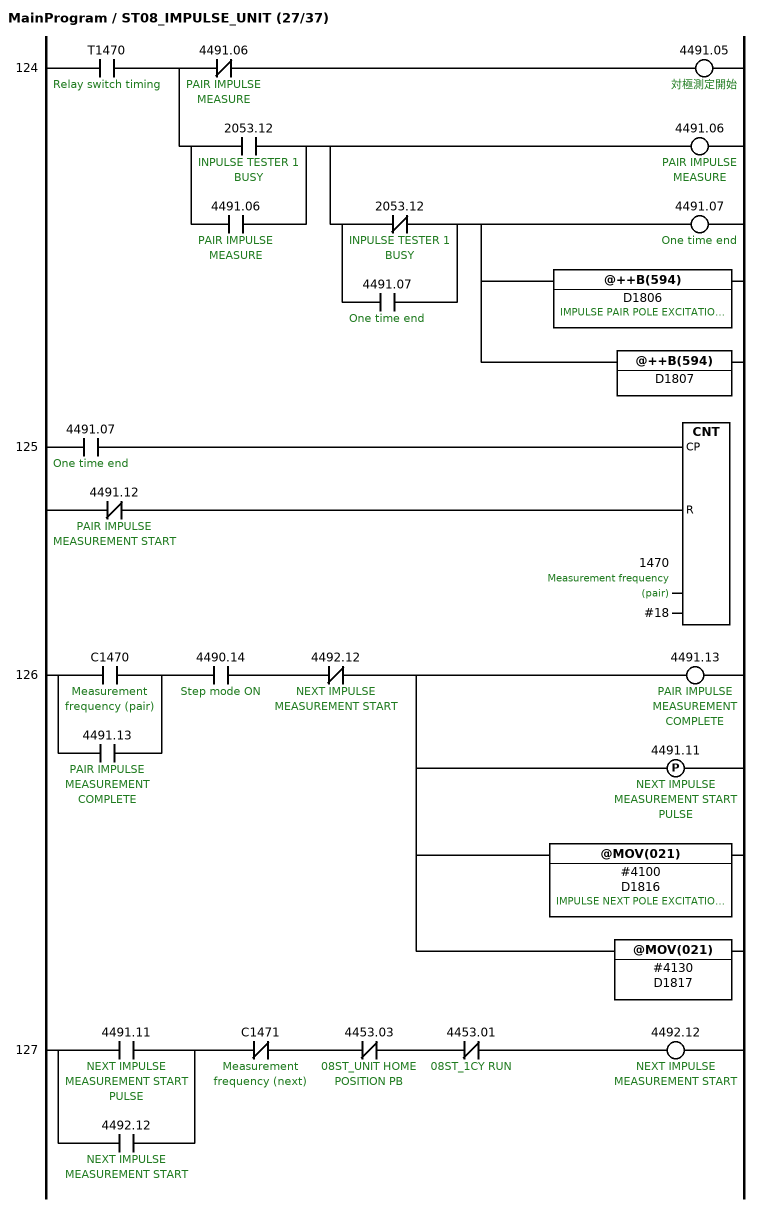
; [picture p456: MainProgram / ST08_IMPULSE_UNIT, rungs 124-127]
; rung 124
LD T1470  ; Relay switch timing
OUT TR0
ANDNOT 4491.06  ; PAIR IMPULSE MEASURE
OUT 4491.05  ; 対極測定開始
LD TR0
LD 2053.12  ; INPULSE TESTER 1 BUSY
OR 4491.06  ; PAIR IMPULSE MEASURE
ANDLD
OUT 4491.06  ; PAIR IMPULSE MEASURE
LDNOT 2053.12  ; INPULSE TESTER 1 BUSY
OR 4491.07  ; One time end
ANDLD
OUT 4491.07  ; One time end
@++B(594) D1806  ; IMPULSE PAIR POLE EXCITATION PATTERN DM STORING(INDIVIDUAL)
@++B(594) D1807
; rung 125
LD 4491.07  ; One time end
LDNOT 4491.12  ; PAIR IMPULSE MEASUREMENT START
CNT 1470 #18  ; Measurement frequency (pair)  // 6 => 18
; rung 126
LD C1470  ; Measurement frequency (pair)
OR 4491.13  ; PAIR IMPULSE MEASUREMENT COMPLETE
AND 4490.14  ; Step mode ON
ANDNOT 4492.12  ; NEXT IMPULSE MEASUREMENT START
OUT 4491.13  ; PAIR IMPULSE MEASUREMENT COMPLETE
DIFU(013) 4491.11  ; NEXT IMPULSE MEASUREMENT START PULSE
@MOV(021) #4100 D1816  ; IMPULSE NEXT POLE EXCITATION PATTERN DM STORING(INDIVIDUAL)
@MOV(021) #4130 D1817
; rung 127
LD 4491.11  ; NEXT IMPULSE MEASUREMENT START PULSE
OR 4492.12  ; NEXT IMPULSE MEASUREMENT START
ANDNOT C1471  ; Measurement frequency (next)
ANDNOT 4453.03  ; 08ST_UNIT HOME POSITION PB
ANDNOT 4453.01  ; 08ST_1CY RUN
OUT 4492.12  ; NEXT IMPULSE MEASUREMENT START

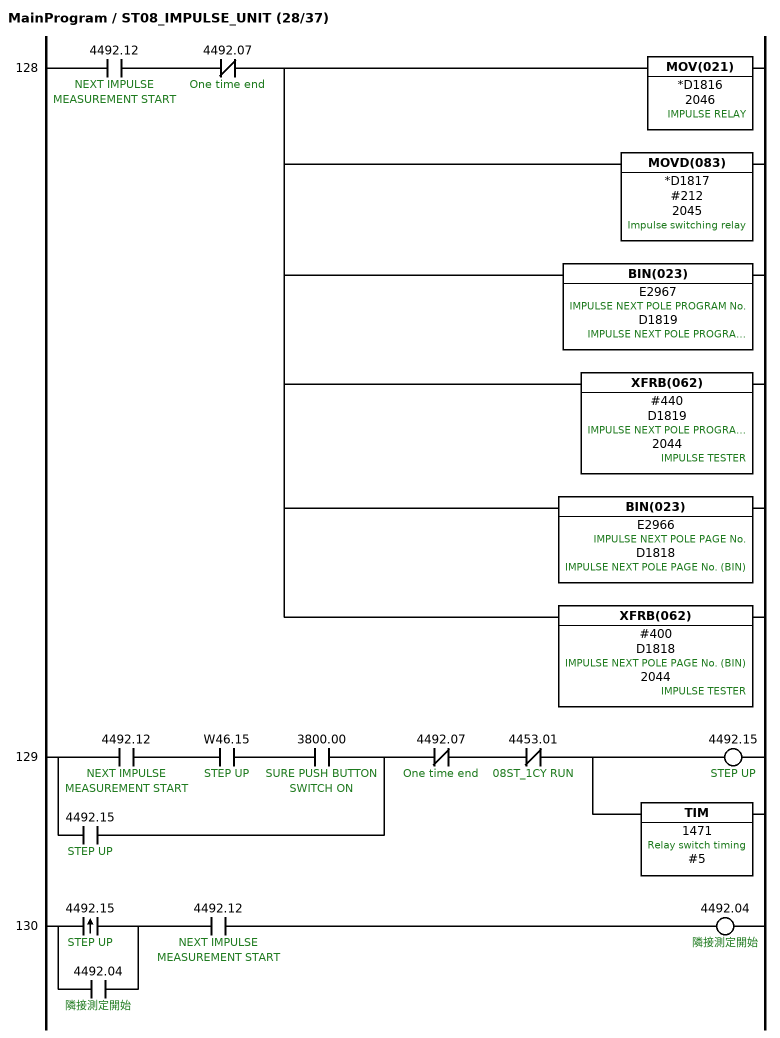
; rung 128
LD 4492.12  ; NEXT IMPULSE MEASUREMENT START
ANDNOT 4492.07  ; One time end
MOV(021) *D1816 2046  ; IMPULSE RELAY
MOVD(083) *D1817 #212 2045  ; Impulse switching relay
BIN(023) E2967 D1819  ; IMPULSE NEXT POLE PROGRAM No., IMPULSE NEXT POLE PROGRAM No.(BIN)
XFRB(062) #440 D1819 2044  ; IMPULSE NEXT POLE PROGRAM No.(BIN), IMPULSE TESTER
BIN(023) E2966 D1818  ; IMPULSE NEXT POLE PAGE No., IMPULSE NEXT POLE PAGE No. (BIN)
XFRB(062) #400 D1818 2044  ; IMPULSE NEXT POLE PAGE No. (BIN), IMPULSE TESTER
; rung 129
LD 4492.12  ; NEXT IMPULSE MEASUREMENT START
AND W46.15  ; STEP UP
AND 3800.00  ; SURE PUSH BUTTON SWITCH ON
OR 4492.15  ; STEP UP
ANDNOT 4492.07  ; One time end
ANDNOT 4453.01  ; 08ST_1CY RUN
OUT 4492.15  ; STEP UP
TIM 1471 #5  ; Relay switch timing
; rung 130
@LD 4492.15  ; STEP UP
OR 4492.04  ; 隣接測定開始
AND 4492.12  ; NEXT IMPULSE MEASUREMENT START
OUT 4492.04  ; 隣接測定開始

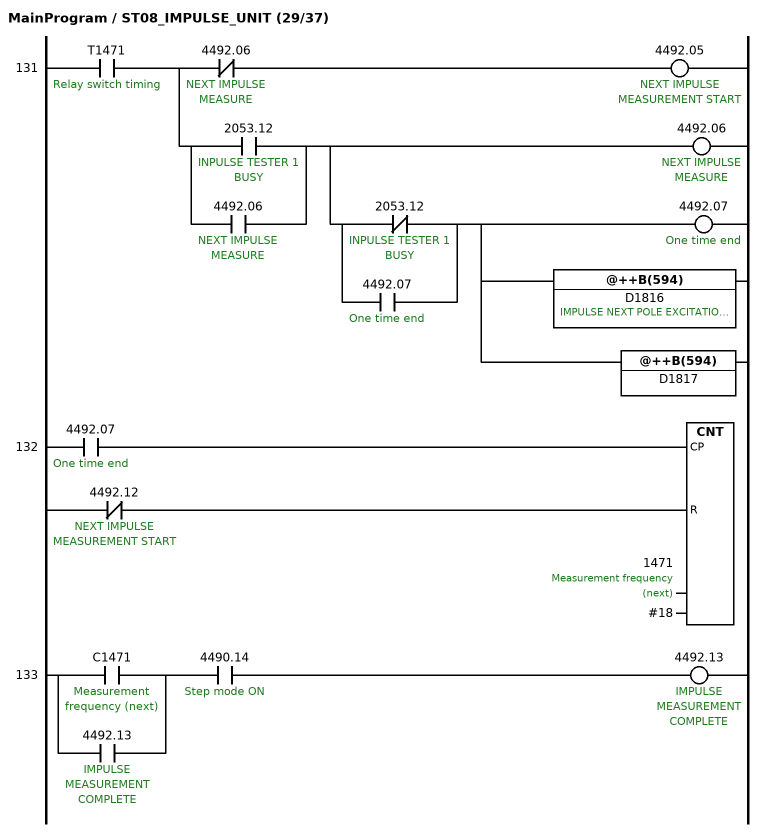
; rung 131
LD T1471  ; Relay switch timing
OUT TR0
ANDNOT 4492.06  ; NEXT IMPULSE MEASURE
OUT 4492.05  ; NEXT IMPULSE MEASUREMENT START
LD TR0
LD 2053.12  ; INPULSE TESTER 1 BUSY
OR 4492.06  ; NEXT IMPULSE MEASURE
ANDLD
OUT 4492.06  ; NEXT IMPULSE MEASURE
LDNOT 2053.12  ; INPULSE TESTER 1 BUSY
OR 4492.07  ; One time end
ANDLD
OUT 4492.07  ; One time end
@++B(594) D1816  ; IMPULSE NEXT POLE EXCITATION PATTERN DM STORING(INDIVIDUAL)
@++B(594) D1817
; rung 132
LD 4492.07  ; One time end
LDNOT 4492.12  ; NEXT IMPULSE MEASUREMENT START
CNT 1471 #18  ; Measurement frequency (next)
; rung 133
LD C1471  ; Measurement frequency (next)
OR 4492.13  ; IMPULSE MEASUREMENT COMPLETE
AND 4490.14  ; Step mode ON
OUT 4492.13  ; IMPULSE MEASUREMENT COMPLETE

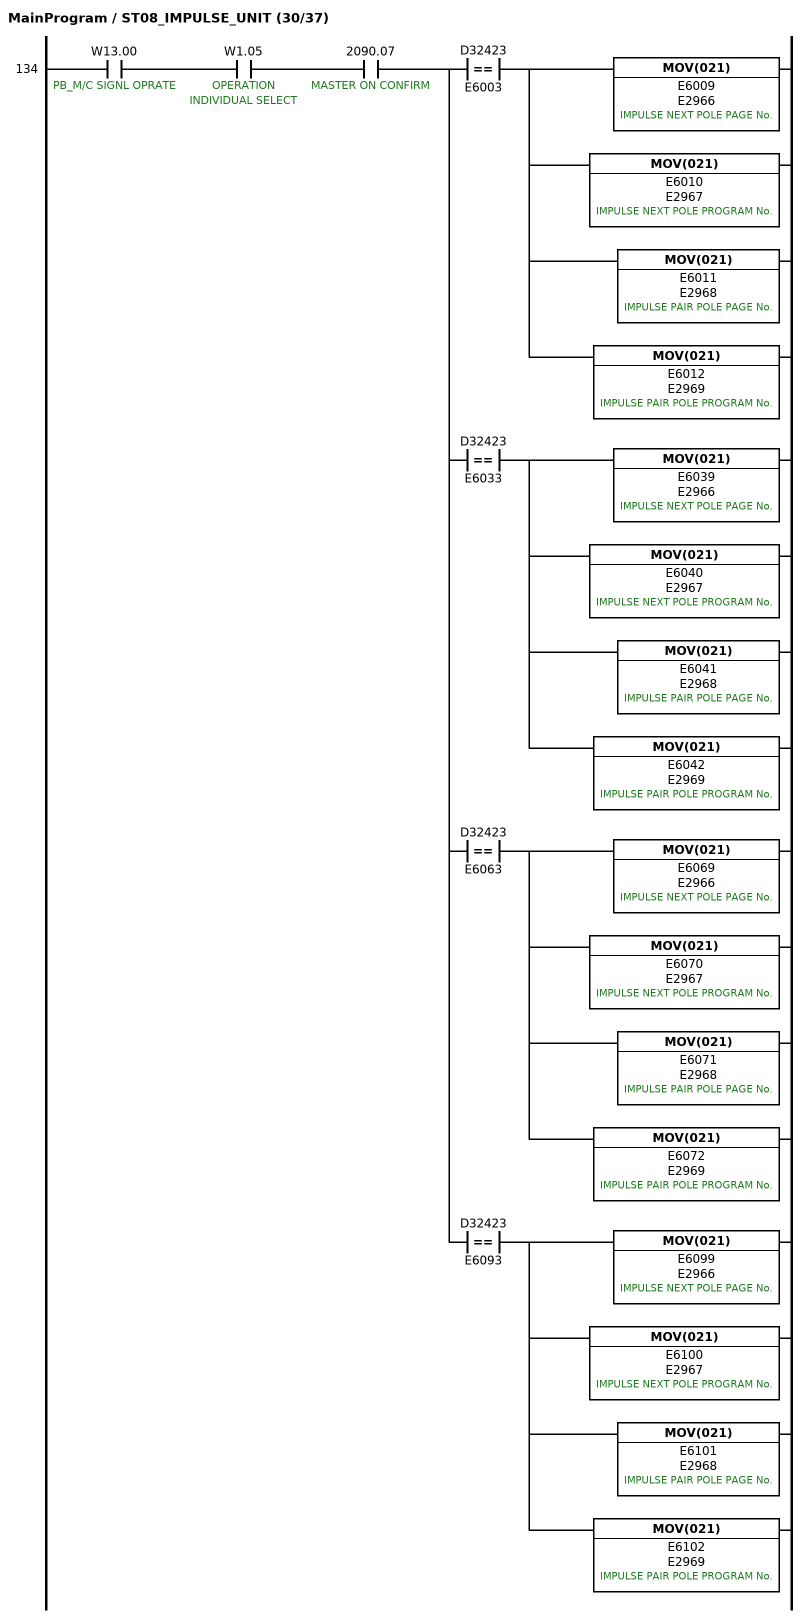
; rung 134
LD W13.00  ; PB_M/C SIGNL OPRATE
AND W1.05  ; OPERATION INDIVIDUAL SELECT
AND 2090.07  ; MASTER ON CONFIRM
OUT TR0
AND=(300) D32423 E6003
MOV(021) E6009 E2966  ; IMPULSE NEXT POLE PAGE No.
MOV(021) E6010 E2967  ; IMPULSE NEXT POLE PROGRAM No.
MOV(021) E6011 E2968  ; IMPULSE PAIR POLE PAGE No.
MOV(021) E6012 E2969  ; IMPULSE PAIR POLE PROGRAM No.
LD TR0
AND=(300) D32423 E6033
MOV(021) E6039 E2966  ; IMPULSE NEXT POLE PAGE No.
MOV(021) E6040 E2967  ; IMPULSE NEXT POLE PROGRAM No.
MOV(021) E6041 E2968  ; IMPULSE PAIR POLE PAGE No.
MOV(021) E6042 E2969  ; IMPULSE PAIR POLE PROGRAM No.
LD TR0
AND=(300) D32423 E6063
MOV(021) E6069 E2966  ; IMPULSE NEXT POLE PAGE No.
MOV(021) E6070 E2967  ; IMPULSE NEXT POLE PROGRAM No.
MOV(021) E6071 E2968  ; IMPULSE PAIR POLE PAGE No.
MOV(021) E6072 E2969  ; IMPULSE PAIR POLE PROGRAM No.
LD TR0
AND=(300) D32423 E6093
MOV(021) E6099 E2966  ; IMPULSE NEXT POLE PAGE No.
MOV(021) E6100 E2967  ; IMPULSE NEXT POLE PROGRAM No.
MOV(021) E6101 E2968  ; IMPULSE PAIR POLE PAGE No.
MOV(021) E6102 E2969  ; IMPULSE PAIR POLE PROGRAM No.

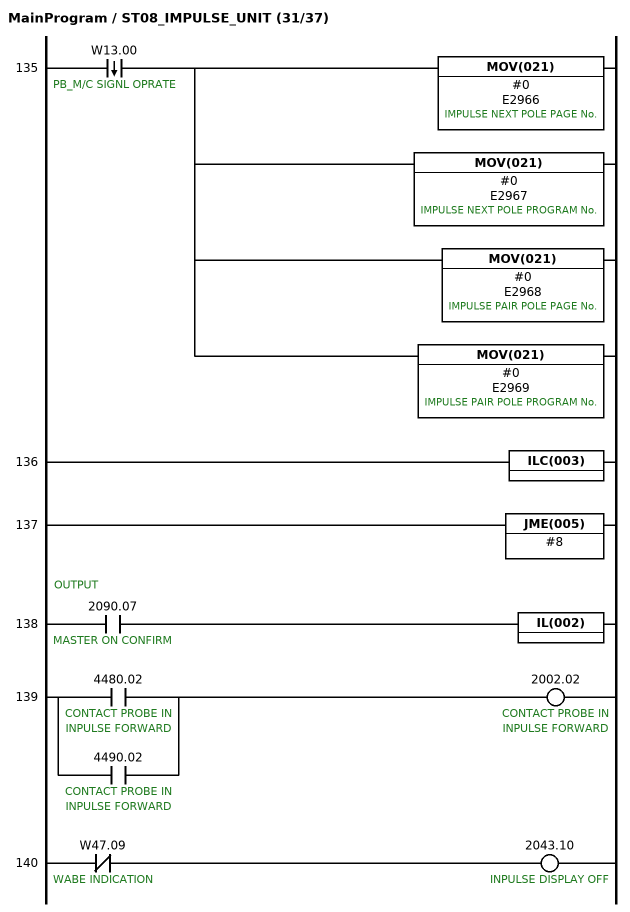
; rung 135
%LD W13.00  ; PB_M/C SIGNL OPRATE
MOV(021) #0 E2966  ; IMPULSE NEXT POLE PAGE No.
MOV(021) #0 E2967  ; IMPULSE NEXT POLE PROGRAM No.
MOV(021) #0 E2968  ; IMPULSE PAIR POLE PAGE No.
MOV(021) #0 E2969  ; IMPULSE PAIR POLE PROGRAM No.
; rung 136
ILC(003)
; rung 137
JME(005) #8
; rung 138: OUTPUT
LD 2090.07  ; MASTER ON CONFIRM
IL(002)
; rung 139
LD 4480.02  ; CONTACT PROBE IN INPULSE FORWARD
OR 4490.02  ; CONTACT PROBE IN INPULSE FORWARD
OUT 2002.02  ; CONTACT PROBE IN INPULSE FORWARD
; rung 140
LDNOT W47.09  ; WABE INDICATION
OUT 2043.10  ; INPULSE DISPLAY OFF

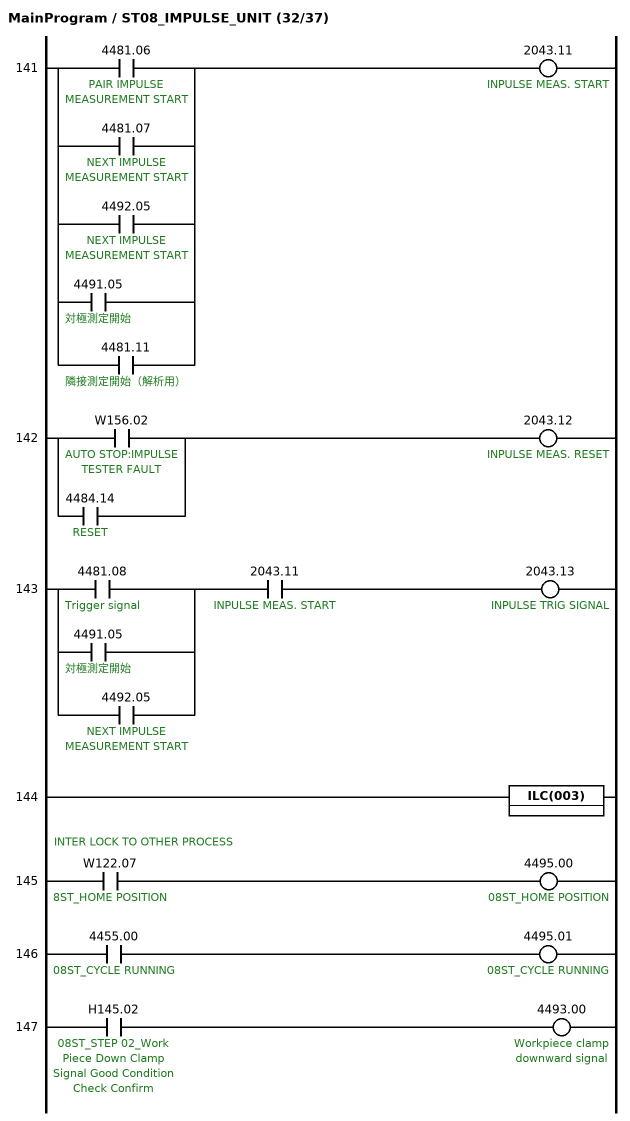
; rung 141
LD 4481.06  ; PAIR IMPULSE MEASUREMENT START
OR 4481.07  ; NEXT IMPULSE MEASUREMENT START
OR 4492.05  ; NEXT IMPULSE MEASUREMENT START
OR 4491.05  ; 対極測定開始
OR 4481.11  ; 隣接測定開始（解析用）
OUT 2043.11  ; INPULSE MEAS. START
; rung 142
LD W156.02  ; AUTO STOP:IMPULSE TESTER FAULT
OR 4484.14  ; RESET
OUT 2043.12  ; INPULSE MEAS. RESET
; rung 143
LD 4481.08  ; Trigger signal
OR 4491.05  ; 対極測定開始
OR 4492.05  ; NEXT IMPULSE MEASUREMENT START
AND 2043.11  ; INPULSE MEAS. START
OUT 2043.13  ; INPULSE TRIG SIGNAL
; rung 144
ILC(003)
; rung 145: INTER LOCK TO OTHER PROCESS
LD W122.07  ; 8ST_HOME POSITION
OUT 4495.00  ; 08ST_HOME POSITION
; rung 146
LD 4455.00  ; 08ST_CYCLE RUNNING
OUT 4495.01  ; 08ST_CYCLE RUNNING
; rung 147
LD H145.02  ; 08ST_STEP 02_Work Piece Down Clamp Signal Good Condition Check Confirm
OUT 4493.00  ; Workpiece clamp downward signal

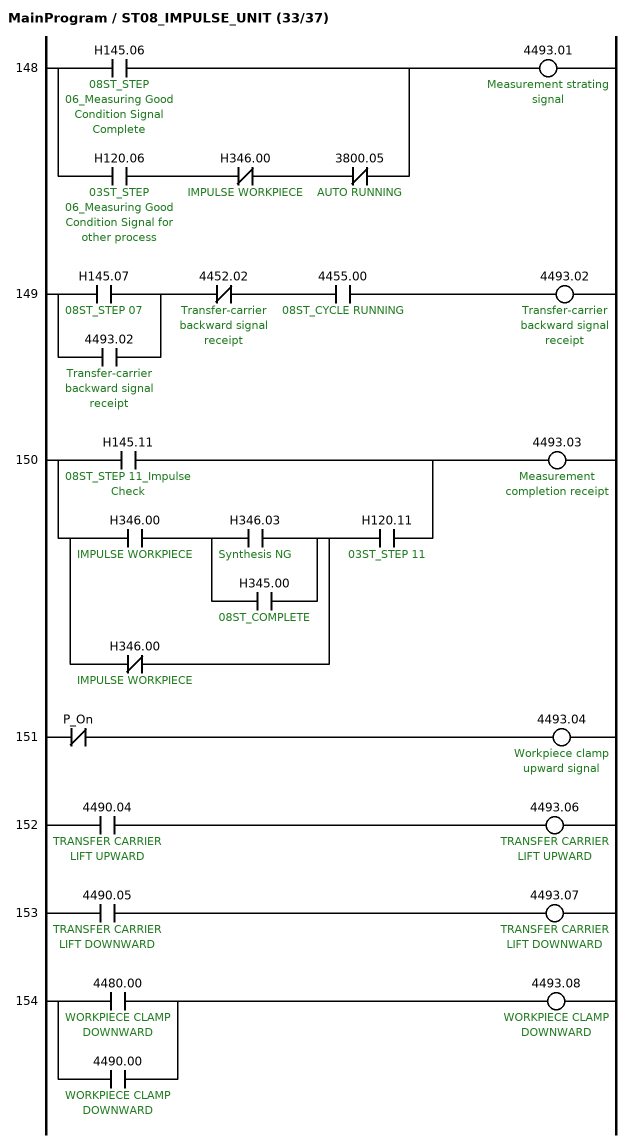
; rung 148
LD H145.06  ; 08ST_STEP 06_Measuring Good Condition Signal Complete
LD H120.06  ; 03ST_STEP 06_Measuring Good Condition Signal for other process
ANDNOT H346.00  ; IMPULSE WORKPIECE
ANDNOT 3800.05  ; AUTO RUNNING
ORLD
OUT 4493.01  ; Measurement strating signal
; rung 149
LD H145.07  ; 08ST_STEP 07
OR 4493.02  ; Transfer-carrier backward signal receipt
ANDNOT 4452.02  ; Transfer-carrier backward signal receipt
AND 4455.00  ; 08ST_CYCLE RUNNING
OUT 4493.02  ; Transfer-carrier backward signal receipt
; rung 150
LD H145.11  ; 08ST_STEP 11_Impulse Check
LD H346.00  ; IMPULSE WORKPIECE
LD H346.03  ; Synthesis NG
OR H345.00  ; 08ST_COMPLETE
ANDLD
ORNOT H346.00  ; IMPULSE WORKPIECE
AND H120.11  ; 03ST_STEP 11
ORLD
OUT 4493.03  ; Measurement completion receipt
; rung 151
LDNOT P_On
OUT 4493.04  ; Workpiece clamp upward signal
; rung 152
LD 4490.04  ; TRANSFER CARRIER LIFT UPWARD
OUT 4493.06  ; TRANSFER CARRIER LIFT UPWARD
; rung 153
LD 4490.05  ; TRANSFER CARRIER LIFT DOWNWARD
OUT 4493.07  ; TRANSFER CARRIER LIFT DOWNWARD
; rung 154
LD 4480.00  ; WORKPIECE CLAMP DOWNWARD
OR 4490.00  ; WORKPIECE CLAMP DOWNWARD
OUT 4493.08  ; WORKPIECE CLAMP DOWNWARD

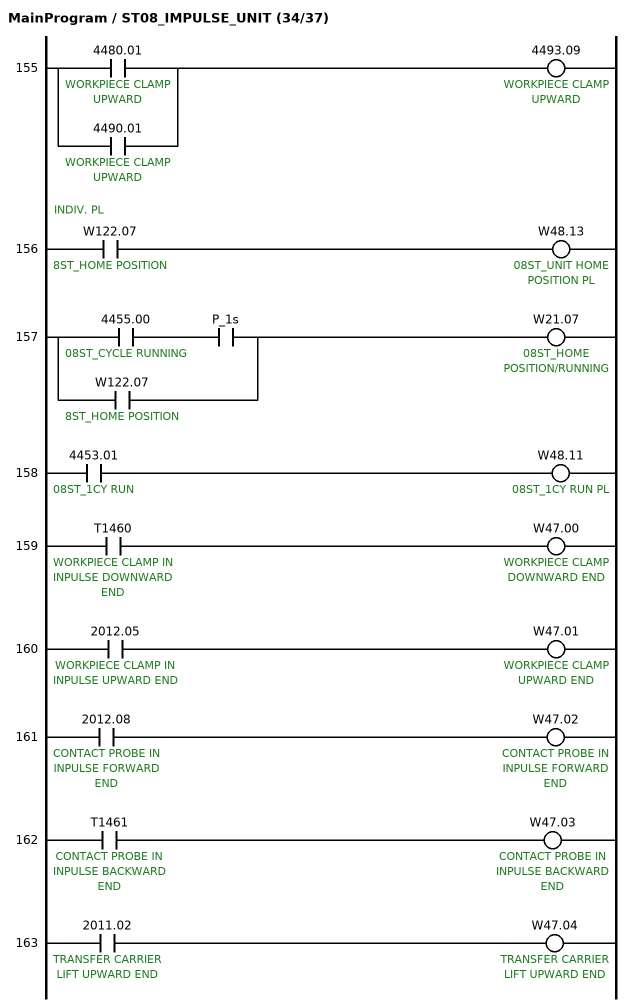
; rung 155
LD 4480.01  ; WORKPIECE CLAMP UPWARD
OR 4490.01  ; WORKPIECE CLAMP UPWARD
OUT 4493.09  ; WORKPIECE CLAMP UPWARD
; rung 156: INDIV. PL
LD W122.07  ; 8ST_HOME POSITION
OUT W48.13  ; 08ST_UNIT HOME POSITION PL
; rung 157
LD 4455.00  ; 08ST_CYCLE RUNNING
AND P_1s
OR W122.07  ; 8ST_HOME POSITION
OUT W21.07  ; 08ST_HOME POSITION/RUNNING
; rung 158
LD 4453.01  ; 08ST_1CY RUN
OUT W48.11  ; 08ST_1CY RUN PL
; rung 159
LD T1460  ; WORKPIECE CLAMP IN INPULSE DOWNWARD END
OUT W47.00  ; WORKPIECE CLAMP DOWNWARD END
; rung 160
LD 2012.05  ; WORKPIECE CLAMP IN INPULSE UPWARD END
OUT W47.01  ; WORKPIECE CLAMP UPWARD END
; rung 161
LD 2012.08  ; CONTACT PROBE IN INPULSE FORWARD END
OUT W47.02  ; CONTACT PROBE IN INPULSE FORWARD END
; rung 162
LD T1461  ; CONTACT PROBE IN INPULSE BACKWARD END
OUT W47.03  ; CONTACT PROBE IN INPULSE BACKWARD END
; rung 163
LD 2011.02  ; TRANSFER CARRIER LIFT UPWARD END
OUT W47.04  ; TRANSFER CARRIER LIFT UPWARD END

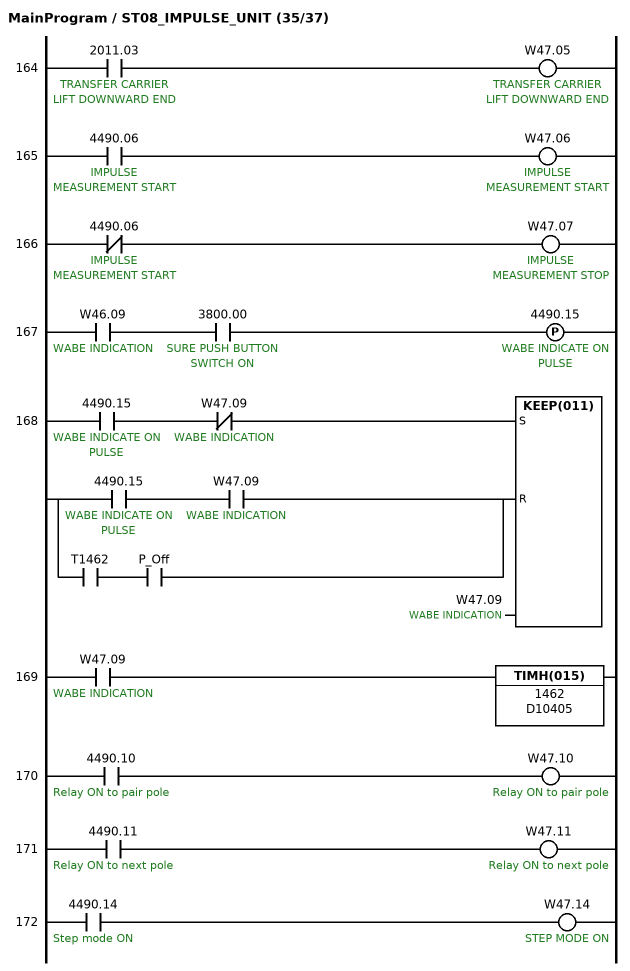
; rung 164
LD 2011.03  ; TRANSFER CARRIER LIFT DOWNWARD END
OUT W47.05  ; TRANSFER CARRIER LIFT DOWNWARD END
; rung 165
LD 4490.06  ; IMPULSE MEASUREMENT START
OUT W47.06  ; IMPULSE MEASUREMENT START
; rung 166
LDNOT 4490.06  ; IMPULSE MEASUREMENT START
OUT W47.07  ; IMPULSE MEASUREMENT STOP
; rung 167
LD W46.09  ; WABE INDICATION
AND 3800.00  ; SURE PUSH BUTTON SWITCH ON
DIFU(013) 4490.15  ; WABE INDICATE ON PULSE
; rung 168
LD 4490.15  ; WABE INDICATE ON PULSE
ANDNOT W47.09  ; WABE INDICATION
LD 4490.15  ; WABE INDICATE ON PULSE
AND W47.09  ; WABE INDICATION
LD T1462
AND P_Off
ORLD
KEEP(011) W47.09  ; WABE INDICATION
; rung 169
LD W47.09  ; WABE INDICATION
TIMH(015) 1462 D10405
; rung 170
LD 4490.10  ; Relay ON to pair pole
OUT W47.10  ; Relay ON to pair pole
; rung 171
LD 4490.11  ; Relay ON to next pole
OUT W47.11  ; Relay ON to next pole
; rung 172
LD 4490.14  ; Step mode ON
OUT W47.14  ; STEP MODE ON

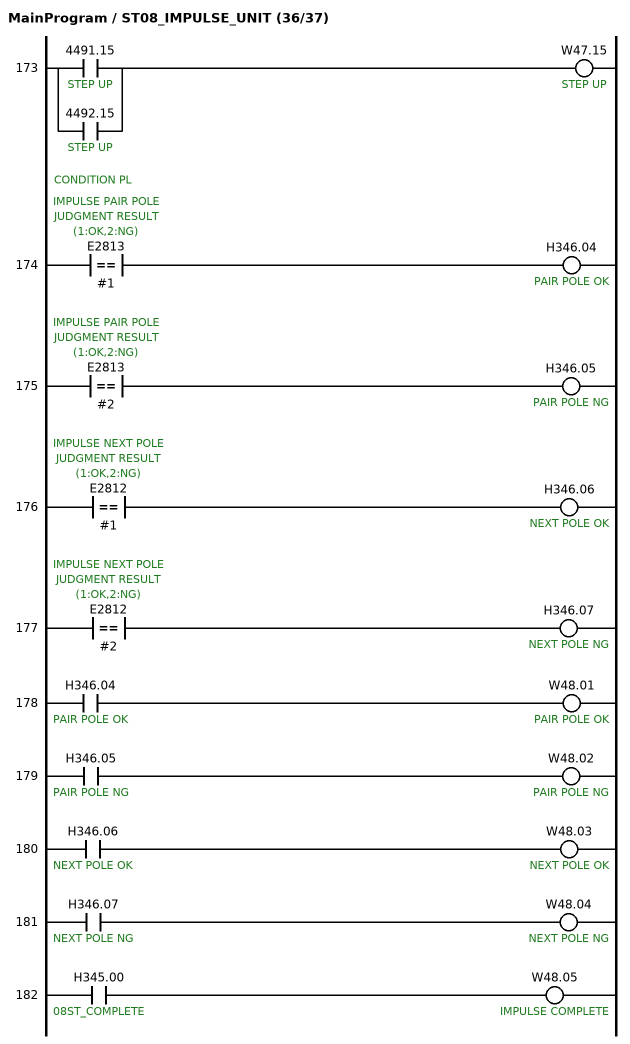
; rung 173
LD 4491.15  ; STEP UP
OR 4492.15  ; STEP UP
OUT W47.15  ; STEP UP
; rung 174: CONDITION PL
LD=(300) E2813 #1  ; IMPULSE PAIR POLE JUDGMENT RESULT (1:OK,2:NG)
OUT H346.04  ; PAIR POLE OK
; rung 175
LD=(300) E2813 #2  ; IMPULSE PAIR POLE JUDGMENT RESULT (1:OK,2:NG)
OUT H346.05  ; PAIR POLE NG
; rung 176
LD=(300) E2812 #1  ; IMPULSE NEXT POLE JUDGMENT RESULT (1:OK,2:NG)
OUT H346.06  ; NEXT POLE OK
; rung 177
LD=(300) E2812 #2  ; IMPULSE NEXT POLE JUDGMENT RESULT (1:OK,2:NG)
OUT H346.07  ; NEXT POLE NG
; rung 178
LD H346.04  ; PAIR POLE OK
OUT W48.01  ; PAIR POLE OK
; rung 179
LD H346.05  ; PAIR POLE NG
OUT W48.02  ; PAIR POLE NG
; rung 180
LD H346.06  ; NEXT POLE OK
OUT W48.03  ; NEXT POLE OK
; rung 181
LD H346.07  ; NEXT POLE NG
OUT W48.04  ; NEXT POLE NG
; rung 182
LD H345.00  ; 08ST_COMPLETE
OUT W48.05  ; IMPULSE COMPLETE

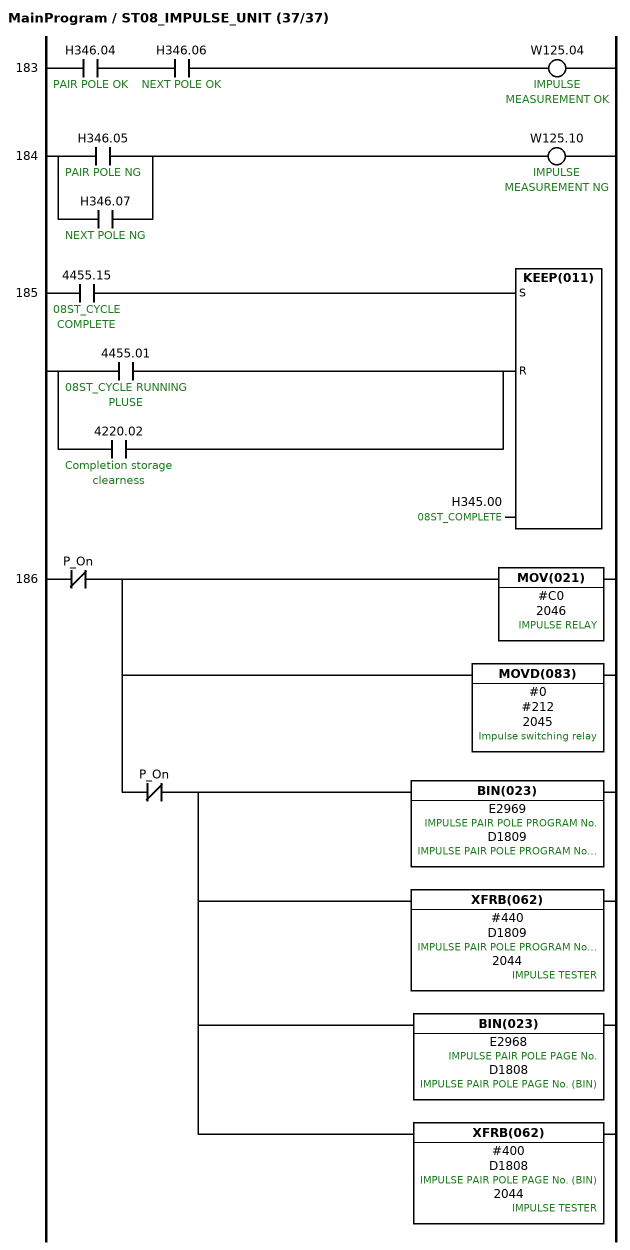
; rung 183
LD H346.04  ; PAIR POLE OK
AND H346.06  ; NEXT POLE OK
OUT W125.04  ; IMPULSE MEASUREMENT OK
; rung 184
LD H346.05  ; PAIR POLE NG
OR H346.07  ; NEXT POLE NG
OUT W125.10  ; IMPULSE MEASUREMENT NG
; rung 185
LD 4455.15  ; 08ST_CYCLE COMPLETE
LD 4455.01  ; 08ST_CYCLE RUNNING PLUSE
OR 4220.02  ; Completion storage clearness
KEEP(011) H345.00  ; 08ST_COMPLETE
; rung 186
LDNOT P_On
MOV(021) #C0 2046  ; IMPULSE RELAY
MOVD(083) #0 #212 2045  ; Impulse switching relay
ANDNOT P_On
BIN(023) E2969 D1809  ; IMPULSE PAIR POLE PROGRAM No., IMPULSE PAIR POLE PROGRAM No. (BIN)
XFRB(062) #440 D1809 2044  ; IMPULSE PAIR POLE PROGRAM No. (BIN), IMPULSE TESTER
BIN(023) E2968 D1808  ; IMPULSE PAIR POLE PAGE No., IMPULSE PAIR POLE PAGE No. (BIN)
XFRB(062) #400 D1808 2044  ; IMPULSE PAIR POLE PAGE No. (BIN), IMPULSE TESTER

### Section ST09_BEARING_INSERT_UNIT

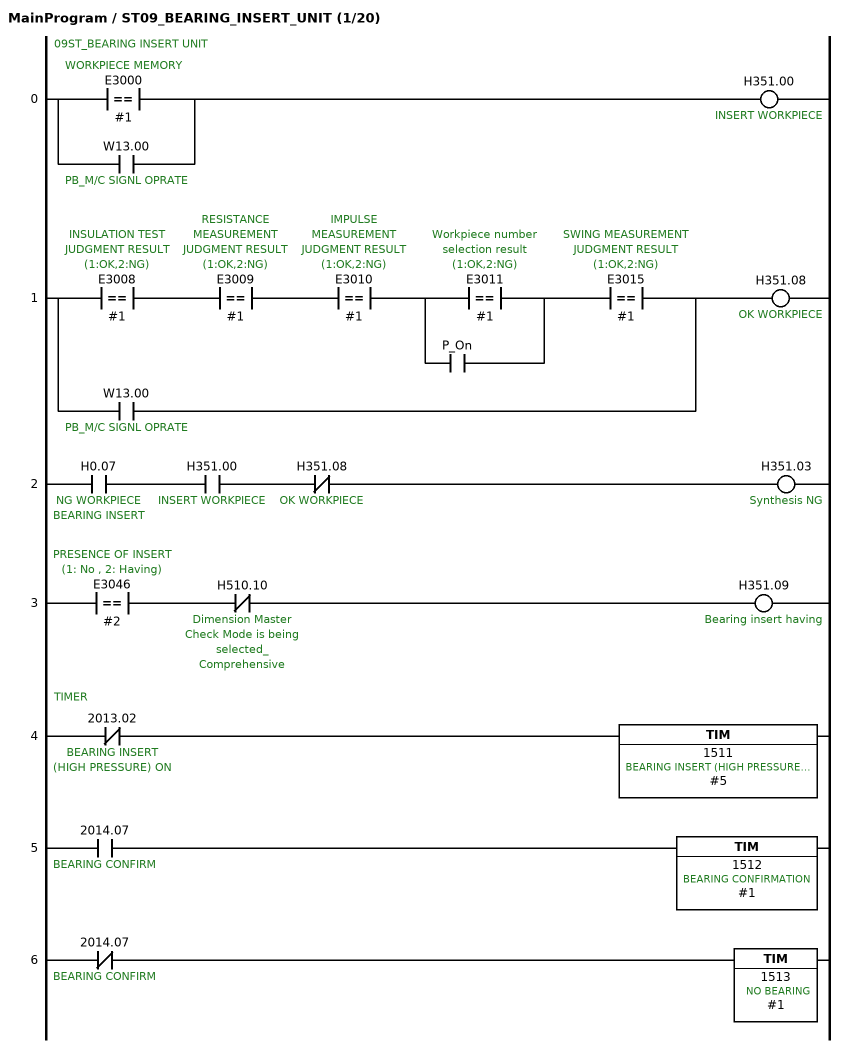
; rung 0: 09ST_BEARING INSERT UNIT
LD=(300) E3000 #1  ; WORKPIECE MEMORY
OR W13.00  ; PB_M/C SIGNL OPRATE
OUT H351.00  ; INSERT WORKPIECE
; rung 1
LD=(300) E3008 #1  ; INSULATION TEST JUDGMENT RESULT (1:OK,2:NG)
AND=(300) E3009 #1  ; RESISTANCE MEASUREMENT JUDGMENT RESULT (1:OK,2:NG)
AND=(300) E3010 #1  ; IMPULSE MEASUREMENT JUDGMENT RESULT (1:OK,2:NG)
LD=(300) E3011 #1  ; Workpiece number selection result (1:OK,2:NG)
OR P_On
ANDLD
AND=(300) E3015 #1  ; SWING MEASUREMENT JUDGMENT RESULT (1:OK,2:NG)
OR W13.00  ; PB_M/C SIGNL OPRATE
OUT H351.08  ; OK WORKPIECE
; rung 2
LD H0.07  ; NG WORKPIECE BEARING INSERT
AND H351.00  ; INSERT WORKPIECE
ANDNOT H351.08  ; OK WORKPIECE
OUT H351.03  ; Synthesis NG
; rung 3
LD=(300) E3046 #2  ; PRESENCE OF INSERT (1: No , 2: Having)
ANDNOT H510.10  ; Dimension Master Check Mode is being selected_Comprehensive
OUT H351.09  ; Bearing insert having
; rung 4: TIMER
LDNOT 2013.02  ; BEARING INSERT (HIGH PRESSURE) ON
TIM 1511 #5  ; BEARING INSERT (HIGH PRESSURE) OFF
; rung 5
LD 2014.07  ; BEARING CONFIRM
TIM 1512 #1  ; BEARING CONFIRMATION
; rung 6
LDNOT 2014.07  ; BEARING CONFIRM
TIM 1513 #1  ; NO BEARING  // #10 => #1

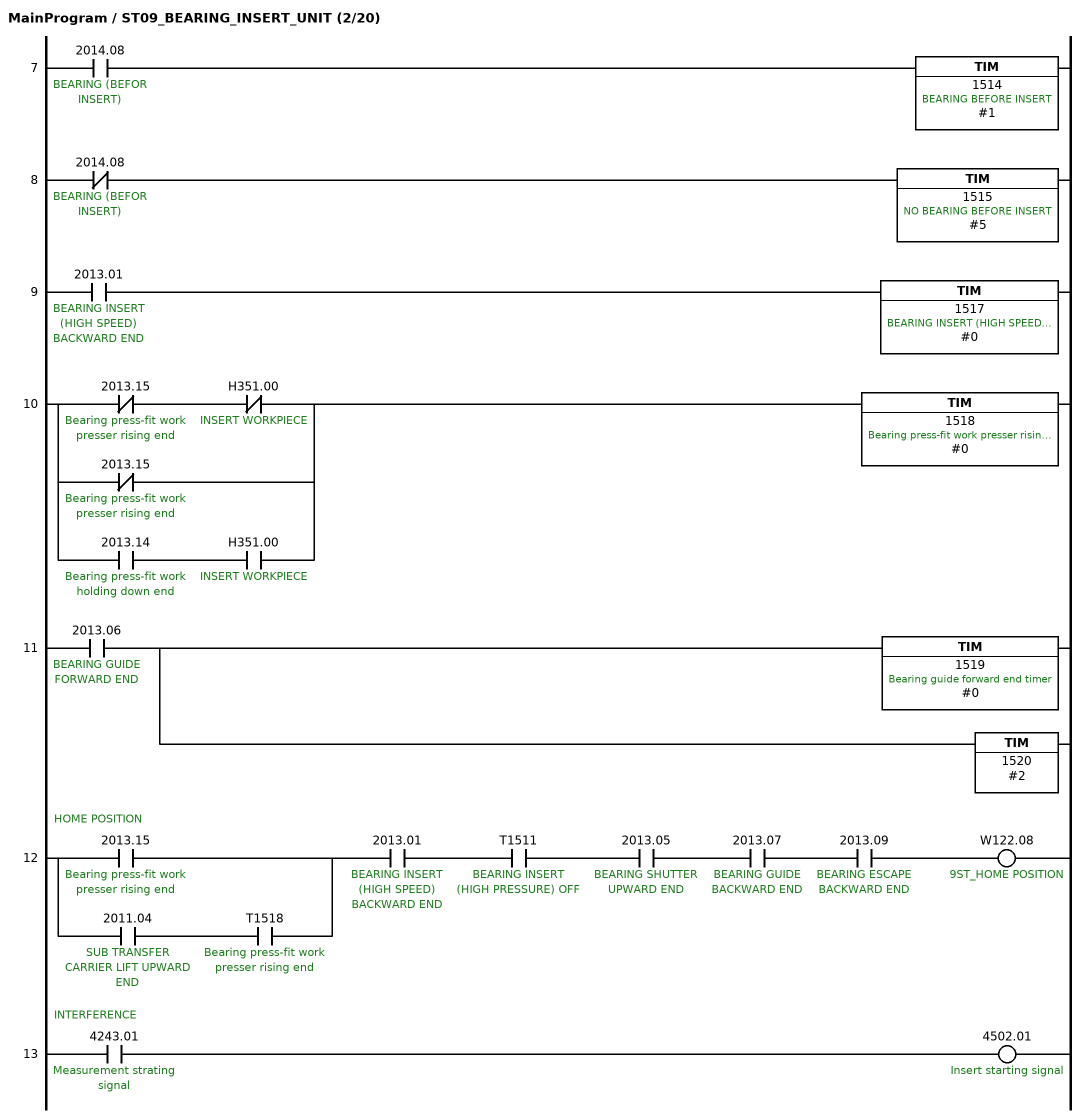
; rung 7
LD 2014.08  ; BEARING (BEFOR INSERT)
TIM 1514 #1  ; BEARING BEFORE INSERT
; rung 8
LDNOT 2014.08  ; BEARING (BEFOR INSERT)
TIM 1515 #5  ; NO BEARING BEFORE INSERT
; rung 9
LD 2013.01  ; BEARING INSERT (HIGH SPEED) BACKWARD END
TIM 1517 #0  ; BEARING INSERT (HIGH SPEED) BACKWARD TIME  // #2 => #0
; rung 10
LDNOT 2013.15  ; Bearing press-fit work presser rising end
ANDNOT H351.00  ; INSERT WORKPIECE
ORNOT 2013.15  ; Bearing press-fit work presser rising end
LD 2013.14  ; Bearing press-fit work holding down end
AND H351.00  ; INSERT WORKPIECE
ORLD
TIM 1518 #0  ; Bearing press-fit work presser rising end
; rung 11
LD 2013.06  ; BEARING GUIDE FORWARD END
TIM 1519 #0  ; Bearing guide forward end timer
TIM 1520 #2
; rung 12: HOME POSITION
LD 2013.15  ; Bearing press-fit work presser rising end
LD 2011.04  ; SUB TRANSFER CARRIER LIFT UPWARD END
AND T1518  ; Bearing press-fit work presser rising end
ORLD
AND 2013.01  ; BEARING INSERT (HIGH SPEED) BACKWARD END
AND T1511  ; BEARING INSERT (HIGH PRESSURE) OFF
AND 2013.05  ; BEARING SHUTTER UPWARD END
AND 2013.07  ; BEARING GUIDE BACKWARD END
AND 2013.09  ; BEARING ESCAPE BACKWARD END
OUT W122.08  ; 9ST_HOME POSITION
; rung 13: INTERFERENCE
LD 4243.01  ; Measurement strating signal
OUT 4502.01  ; Insert starting signal

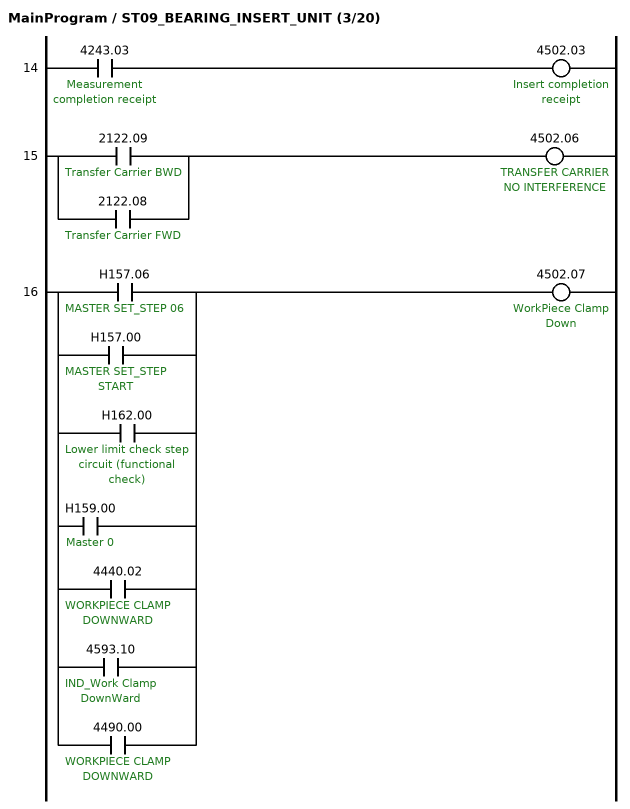
; rung 14
LD 4243.03  ; Measurement completion receipt
OUT 4502.03  ; Insert completion receipt
; rung 15
LD 2122.09  ; Transfer Carrier BWD
OR 2122.08  ; Transfer Carrier FWD
OUT 4502.06  ; TRANSFER CARRIER NO INTERFERENCE
; rung 16
LD H157.06  ; MASTER SET_STEP 06
OR H157.00  ; MASTER SET_STEP START
OR H162.00  ; Lower limit check step circuit (functional check)
OR H159.00  ; Master 0
OR 4440.02  ; WORKPIECE CLAMP DOWNWARD
OR 4593.10  ; IND_Work Clamp DownWard
OR 4490.00  ; WORKPIECE CLAMP DOWNWARD
OUT 4502.07  ; WorkPiece Clamp Down

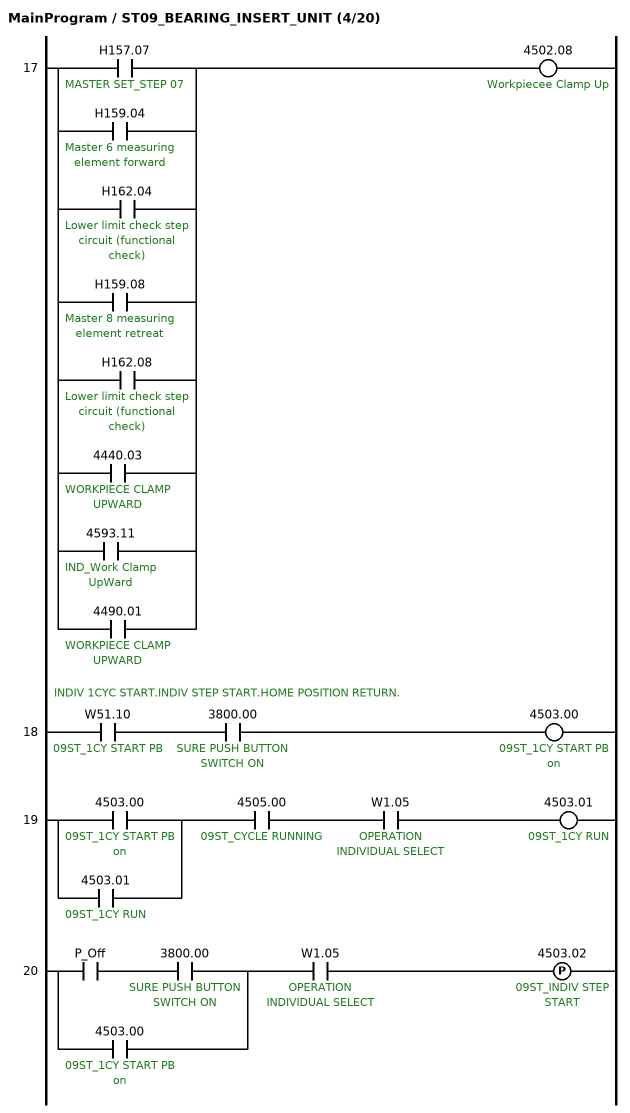
; rung 17
LD H157.07  ; MASTER SET_STEP 07
OR H159.04  ; Master 6 measuring element forward
OR H162.04  ; Lower limit check step circuit (functional check)
OR H159.08  ; Master 8 measuring element retreat
OR H162.08  ; Lower limit check step circuit (functional check)
OR 4440.03  ; WORKPIECE CLAMP UPWARD
OR 4593.11  ; IND_Work Clamp UpWard
OR 4490.01  ; WORKPIECE CLAMP UPWARD
OUT 4502.08  ; Workpiecee Clamp Up
; rung 18: INDIV 1CYC START.INDIV STEP START.HOME POSITION RETURN.
LD W51.10  ; 09ST_1CY START PB
AND 3800.00  ; SURE PUSH BUTTON SWITCH ON
OUT 4503.00  ; 09ST_1CY START PB on
; rung 19
LD 4503.00  ; 09ST_1CY START PB on
OR 4503.01  ; 09ST_1CY RUN
AND 4505.00  ; 09ST_CYCLE RUNNING
AND W1.05  ; OPERATION INDIVIDUAL SELECT
OUT 4503.01  ; 09ST_1CY RUN
; rung 20
LD P_Off
AND 3800.00  ; SURE PUSH BUTTON SWITCH ON
OR 4503.00  ; 09ST_1CY START PB on
AND W1.05  ; OPERATION INDIVIDUAL SELECT
DIFU(013) 4503.02  ; 09ST_INDIV STEP START

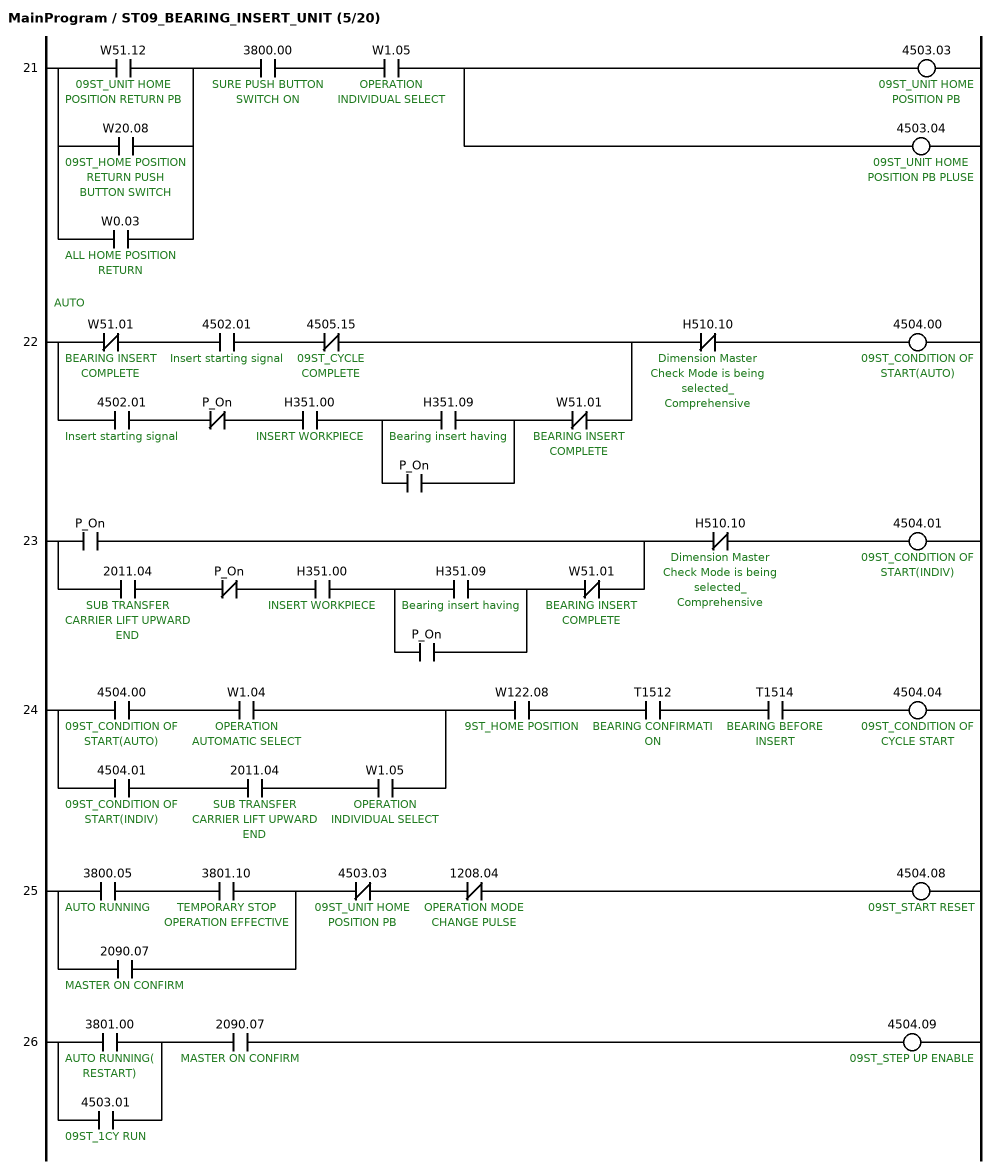
; rung 21
LD W51.12  ; 09ST_UNIT HOME POSITION RETURN PB
OR W20.08  ; 09ST_HOME POSITION RETURN PUSH BUTTON SWITCH
OR W0.03  ; ALL HOME POSITION RETURN
AND 3800.00  ; SURE PUSH BUTTON SWITCH ON
AND W1.05  ; OPERATION INDIVIDUAL SELECT
OUT 4503.03  ; 09ST_UNIT HOME POSITION PB
OUT 4503.04  ; 09ST_UNIT HOME POSITION PB PLUSE
; rung 22: AUTO
LDNOT W51.01  ; BEARING INSERT COMPLETE
AND 4502.01  ; Insert starting signal
ANDNOT 4505.15  ; 09ST_CYCLE COMPLETE
LD 4502.01  ; Insert starting signal
ANDNOT P_On
AND H351.00  ; INSERT WORKPIECE
LD H351.09  ; Bearing insert having
OR P_On
ANDLD
ANDNOT W51.01  ; BEARING INSERT COMPLETE
ORLD
ANDNOT H510.10  ; Dimension Master Check Mode is being selected_Comprehensive
OUT 4504.00  ; 09ST_CONDITION OF START(AUTO)
; rung 23
LD P_On
LD 2011.04  ; SUB TRANSFER CARRIER LIFT UPWARD END
ANDNOT P_On
AND H351.00  ; INSERT WORKPIECE
LD H351.09  ; Bearing insert having
OR P_On
ANDLD
ANDNOT W51.01  ; BEARING INSERT COMPLETE
ORLD
ANDNOT H510.10  ; Dimension Master Check Mode is being selected_Comprehensive
OUT 4504.01  ; 09ST_CONDITION OF START(INDIV)
; rung 24
LD 4504.00  ; 09ST_CONDITION OF START(AUTO)
AND W1.04  ; OPERATION AUTOMATIC SELECT
LD 4504.01  ; 09ST_CONDITION OF START(INDIV)
AND 2011.04  ; SUB TRANSFER CARRIER LIFT UPWARD END
AND W1.05  ; OPERATION INDIVIDUAL SELECT
ORLD
AND W122.08  ; 9ST_HOME POSITION
AND T1512  ; BEARING CONFIRMATION
AND T1514  ; BEARING BEFORE INSERT
OUT 4504.04  ; 09ST_CONDITION OF CYCLE START
; rung 25
LD 3800.05  ; AUTO RUNNING
AND 3801.10  ; TEMPORARY STOP OPERATION EFFECTIVE
OR 2090.07  ; MASTER ON CONFIRM
ANDNOT 4503.03  ; 09ST_UNIT HOME POSITION PB
ANDNOT 1208.04  ; OPERATION MODE CHANGE PULSE
OUT 4504.08  ; 09ST_START RESET
; rung 26
LD 3801.00  ; AUTO RUNNING(RESTART)
OR 4503.01  ; 09ST_1CY RUN
AND 2090.07  ; MASTER ON CONFIRM
OUT 4504.09  ; 09ST_STEP UP ENABLE

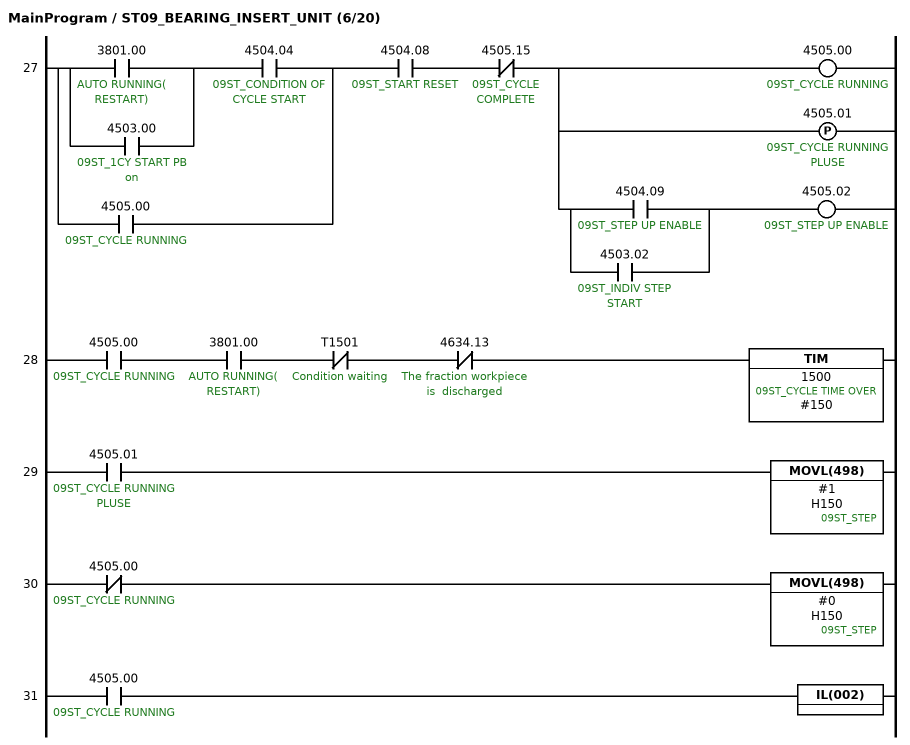
; rung 27
LD 3801.00  ; AUTO RUNNING(RESTART)
OR 4503.00  ; 09ST_1CY START PB on
AND 4504.04  ; 09ST_CONDITION OF CYCLE START
OR 4505.00  ; 09ST_CYCLE RUNNING
AND 4504.08  ; 09ST_START RESET
ANDNOT 4505.15  ; 09ST_CYCLE COMPLETE
OUT 4505.00  ; 09ST_CYCLE RUNNING
DIFU(013) 4505.01  ; 09ST_CYCLE RUNNING PLUSE
LD 4504.09  ; 09ST_STEP UP ENABLE
OR 4503.02  ; 09ST_INDIV STEP START
ANDLD
OUT 4505.02  ; 09ST_STEP UP ENABLE
; rung 28
LD 4505.00  ; 09ST_CYCLE RUNNING
AND 3801.00  ; AUTO RUNNING(RESTART)
ANDNOT T1501  ; Condition waiting
ANDNOT 4634.13  ; The fraction workpiece is  discharged
TIM 1500 #150  ; 09ST_CYCLE TIME OVER
; rung 29
LD 4505.01  ; 09ST_CYCLE RUNNING PLUSE
MOVL(498) #1 H150  ; 09ST_STEP
; rung 30
LDNOT 4505.00  ; 09ST_CYCLE RUNNING
MOVL(498) #0 H150  ; 09ST_STEP
; rung 31
LD 4505.00  ; 09ST_CYCLE RUNNING
IL(002)

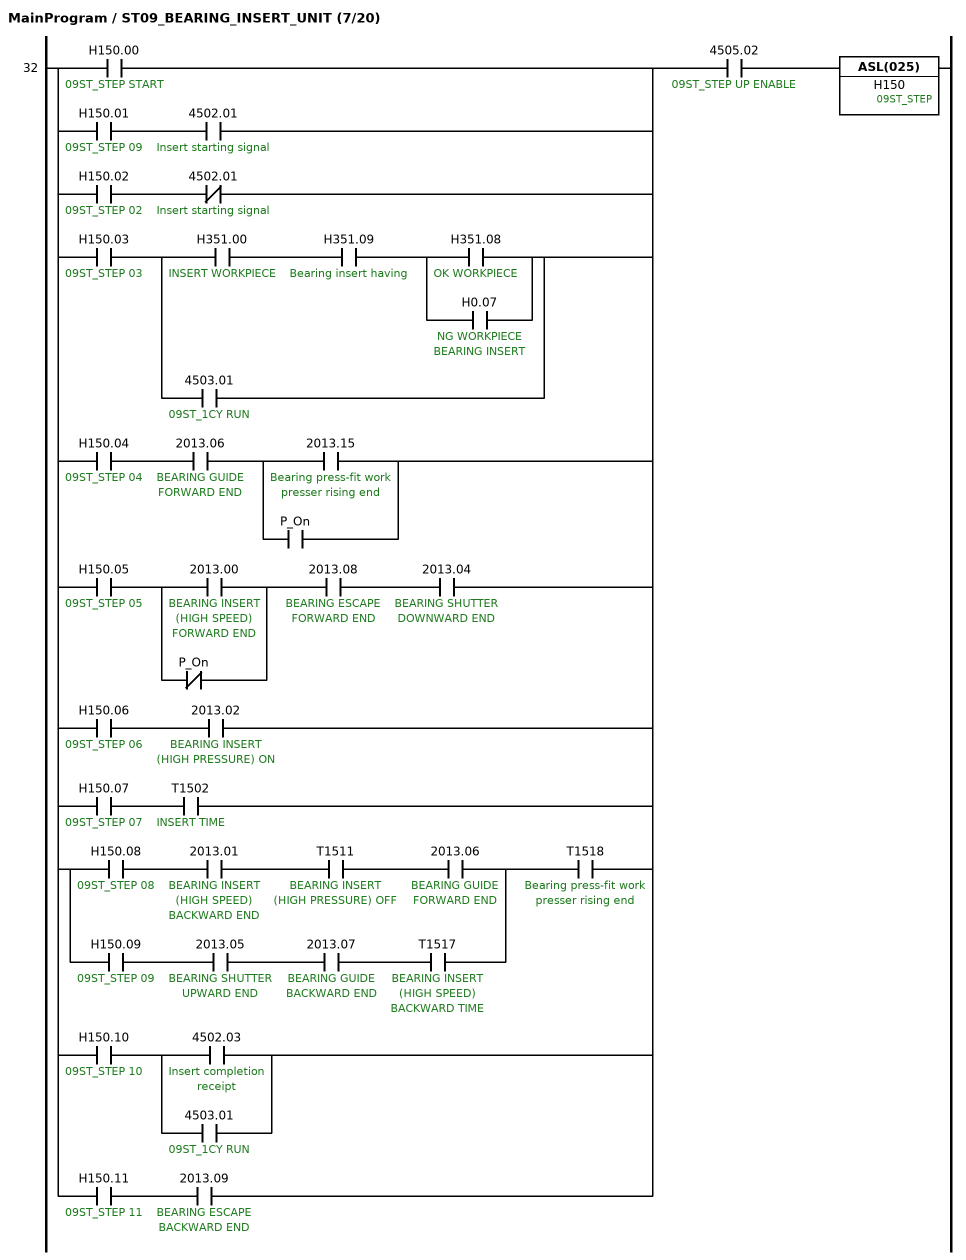
; rung 32
LD H150.00  ; 09ST_STEP START
LD H150.01  ; 09ST_STEP 09
AND 4502.01  ; Insert starting signal
ORLD
LD H150.02  ; 09ST_STEP 02
ANDNOT 4502.01  ; Insert starting signal
ORLD
LD H150.03  ; 09ST_STEP 03
LD H351.00  ; INSERT WORKPIECE
AND H351.09  ; Bearing insert having
LD H351.08  ; OK WORKPIECE
OR H0.07  ; NG WORKPIECE BEARING INSERT
ANDLD
OR 4503.01  ; 09ST_1CY RUN
ANDLD
ORLD
LD H150.04  ; 09ST_STEP 04
AND 2013.06  ; BEARING GUIDE FORWARD END
LD 2013.15  ; Bearing press-fit work presser rising end
OR P_On
ANDLD
ORLD
LD H150.05  ; 09ST_STEP 05
LD 2013.00  ; BEARING INSERT (HIGH SPEED) FORWARD END
ORNOT P_On
ANDLD
AND 2013.08  ; BEARING ESCAPE FORWARD END
AND 2013.04  ; BEARING SHUTTER DOWNWARD END
ORLD
LD H150.06  ; 09ST_STEP 06
AND 2013.02  ; BEARING INSERT (HIGH PRESSURE) ON
ORLD
LD H150.07  ; 09ST_STEP 07
AND T1502  ; INSERT TIME
ORLD
LD H150.08  ; 09ST_STEP 08
AND 2013.01  ; BEARING INSERT (HIGH SPEED) BACKWARD END
AND T1511  ; BEARING INSERT (HIGH PRESSURE) OFF
AND 2013.06  ; BEARING GUIDE FORWARD END
LD H150.09  ; 09ST_STEP 09
AND 2013.05  ; BEARING SHUTTER UPWARD END
AND 2013.07  ; BEARING GUIDE BACKWARD END
AND T1517  ; BEARING INSERT (HIGH SPEED) BACKWARD TIME
ORLD
AND T1518  ; Bearing press-fit work presser rising end
ORLD
LD H150.10  ; 09ST_STEP 10
LD 4502.03  ; Insert completion receipt
OR 4503.01  ; 09ST_1CY RUN
ANDLD
ORLD
LD H150.11  ; 09ST_STEP 11
AND 2013.09  ; BEARING ESCAPE BACKWARD END
ORLD
AND 4505.02  ; 09ST_STEP UP ENABLE
ASL(025) H150  ; 09ST_STEP

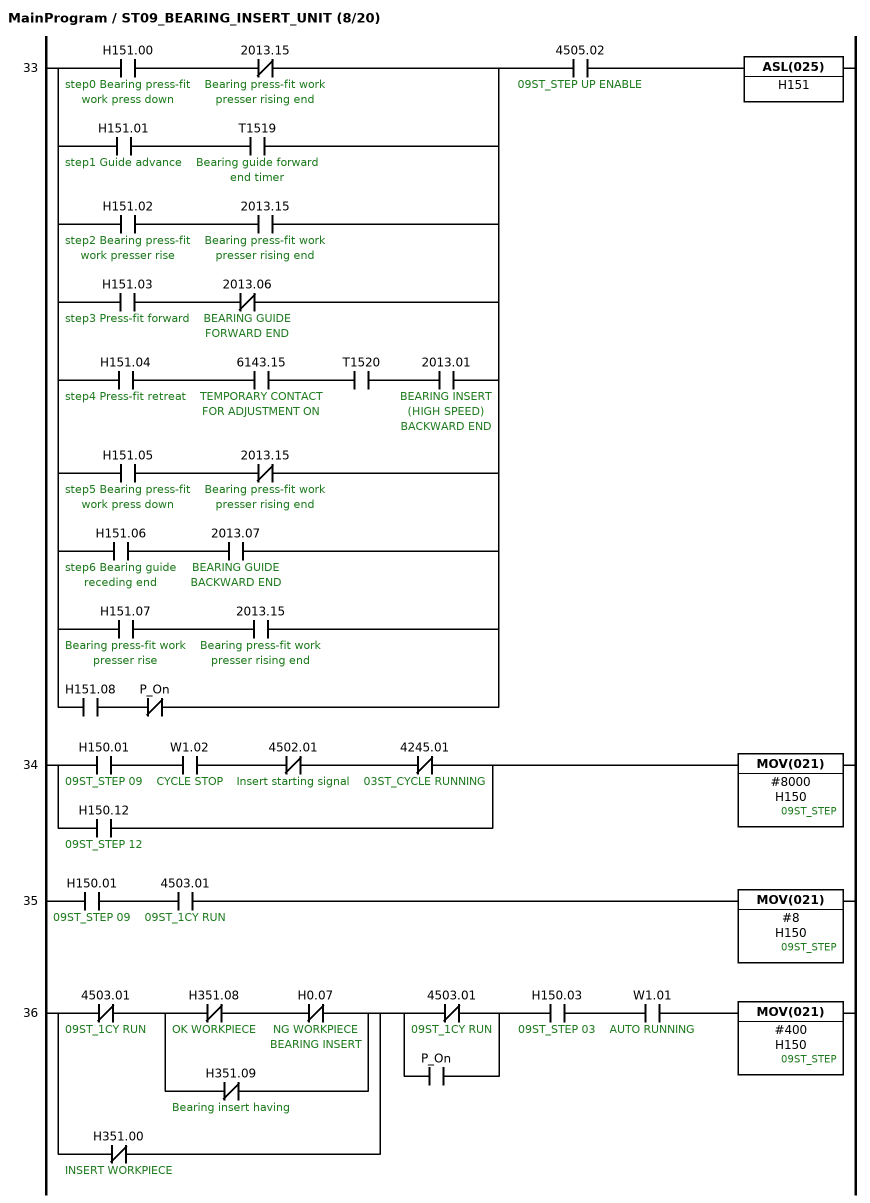
; rung 33
LD H151.00  ; step0 Bearing press-fit work press down
ANDNOT 2013.15  ; Bearing press-fit work presser rising end
LD H151.01  ; step1 Guide advance
AND T1519  ; Bearing guide forward end timer
ORLD
LD H151.02  ; step2 Bearing press-fit work presser rise
AND 2013.15  ; Bearing press-fit work presser rising end
ORLD
LD H151.03  ; step3 Press-fit forward
ANDNOT 2013.06  ; BEARING GUIDE FORWARD END
ORLD
LD H151.04  ; step4 Press-fit retreat
AND 6143.15  ; TEMPORARY CONTACT FOR ADJUSTMENT ON
AND T1520
AND 2013.01  ; BEARING INSERT (HIGH SPEED) BACKWARD END
ORLD
LD H151.05  ; step5 Bearing press-fit work press down
ANDNOT 2013.15  ; Bearing press-fit work presser rising end
ORLD
LD H151.06  ; step6 Bearing guide receding end
AND 2013.07  ; BEARING GUIDE BACKWARD END
ORLD
LD H151.07  ; Bearing press-fit work presser rise
AND 2013.15  ; Bearing press-fit work presser rising end
ORLD
LD H151.08
ANDNOT P_On
ORLD
AND 4505.02  ; 09ST_STEP UP ENABLE
ASL(025) H151
; rung 34
LD H150.01  ; 09ST_STEP 09
AND W1.02  ; CYCLE STOP
ANDNOT 4502.01  ; Insert starting signal
ANDNOT 4245.01  ; 03ST_CYCLE RUNNING
OR H150.12  ; 09ST_STEP 12
MOV(021) #8000 H150  ; 09ST_STEP
; rung 35
LD H150.01  ; 09ST_STEP 09
AND 4503.01  ; 09ST_1CY RUN
MOV(021) #8 H150  ; 09ST_STEP
; rung 36
LDNOT 4503.01  ; 09ST_1CY RUN
LDNOT H351.08  ; OK WORKPIECE
ANDNOT H0.07  ; NG WORKPIECE BEARING INSERT
ORNOT H351.09  ; Bearing insert having
ANDLD
ORNOT H351.00  ; INSERT WORKPIECE
LDNOT 4503.01  ; 09ST_1CY RUN
OR P_On
ANDLD
AND H150.03  ; 09ST_STEP 03
AND W1.01  ; AUTO RUNNING
MOV(021) #400 H150  ; 09ST_STEP

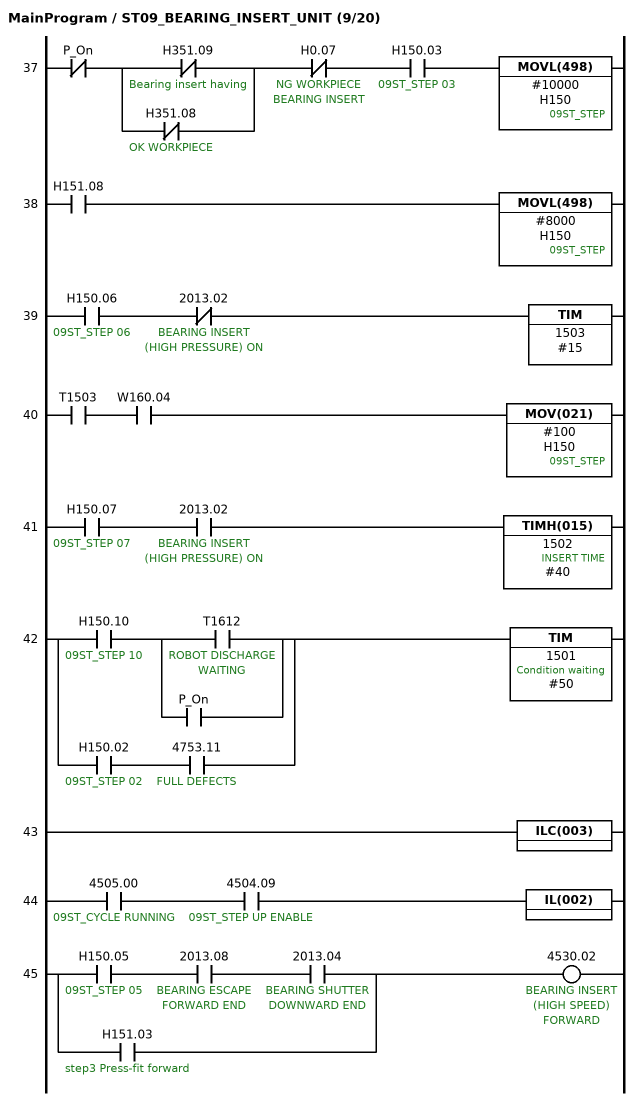
; rung 37
LDNOT P_On
LDNOT H351.09  ; Bearing insert having
ORNOT H351.08  ; OK WORKPIECE
ANDLD
ANDNOT H0.07  ; NG WORKPIECE BEARING INSERT
AND H150.03  ; 09ST_STEP 03
MOVL(498) #10000 H150  ; 09ST_STEP
; rung 38
LD H151.08
MOVL(498) #8000 H150  ; 09ST_STEP
; rung 39
LD H150.06  ; 09ST_STEP 06
ANDNOT 2013.02  ; BEARING INSERT (HIGH PRESSURE) ON
TIM 1503 #15
; rung 40
LD T1503
AND W160.04
MOV(021) #100 H150  ; 09ST_STEP
; rung 41
LD H150.07  ; 09ST_STEP 07
AND 2013.02  ; BEARING INSERT (HIGH PRESSURE) ON
TIMH(015) 1502 #40  ; INSERT TIME  // #125 => #40
; rung 42
LD H150.10  ; 09ST_STEP 10
LD T1612  ; ROBOT DISCHARGE WAITING
OR P_On
ANDLD
LD H150.02  ; 09ST_STEP 02
AND 4753.11  ; FULL DEFECTS
ORLD
TIM 1501 #50  ; Condition waiting
; rung 43
ILC(003)
; rung 44
LD 4505.00  ; 09ST_CYCLE RUNNING
AND 4504.09  ; 09ST_STEP UP ENABLE
IL(002)
; rung 45
LD H150.05  ; 09ST_STEP 05
AND 2013.08  ; BEARING ESCAPE FORWARD END
AND 2013.04  ; BEARING SHUTTER DOWNWARD END
OR H151.03  ; step3 Press-fit forward
OUT 4530.02  ; BEARING INSERT (HIGH SPEED) FORWARD

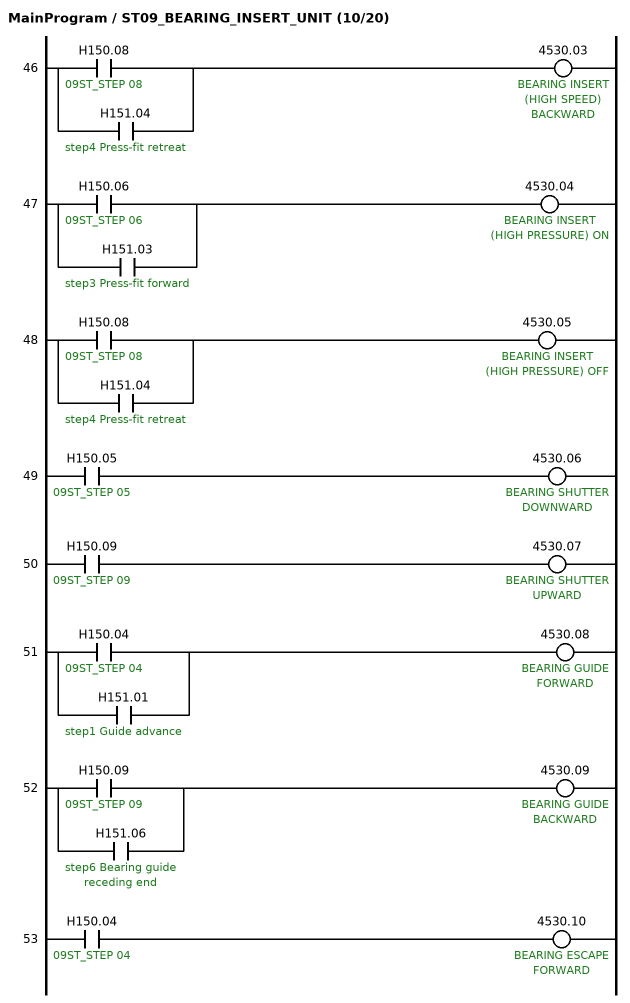
; rung 46
LD H150.08  ; 09ST_STEP 08
OR H151.04  ; step4 Press-fit retreat
OUT 4530.03  ; BEARING INSERT (HIGH SPEED) BACKWARD
; rung 47
LD H150.06  ; 09ST_STEP 06
OR H151.03  ; step3 Press-fit forward
OUT 4530.04  ; BEARING INSERT (HIGH PRESSURE) ON
; rung 48
LD H150.08  ; 09ST_STEP 08
OR H151.04  ; step4 Press-fit retreat
OUT 4530.05  ; BEARING INSERT (HIGH PRESSURE) OFF
; rung 49
LD H150.05  ; 09ST_STEP 05
OUT 4530.06  ; BEARING SHUTTER DOWNWARD
; rung 50
LD H150.09  ; 09ST_STEP 09
OUT 4530.07  ; BEARING SHUTTER UPWARD
; rung 51
LD H150.04  ; 09ST_STEP 04
OR H151.01  ; step1 Guide advance
OUT 4530.08  ; BEARING GUIDE FORWARD
; rung 52
LD H150.09  ; 09ST_STEP 09
OR H151.06  ; step6 Bearing guide receding end
OUT 4530.09  ; BEARING GUIDE BACKWARD
; rung 53
LD H150.04  ; 09ST_STEP 04
OUT 4530.10  ; BEARING ESCAPE FORWARD

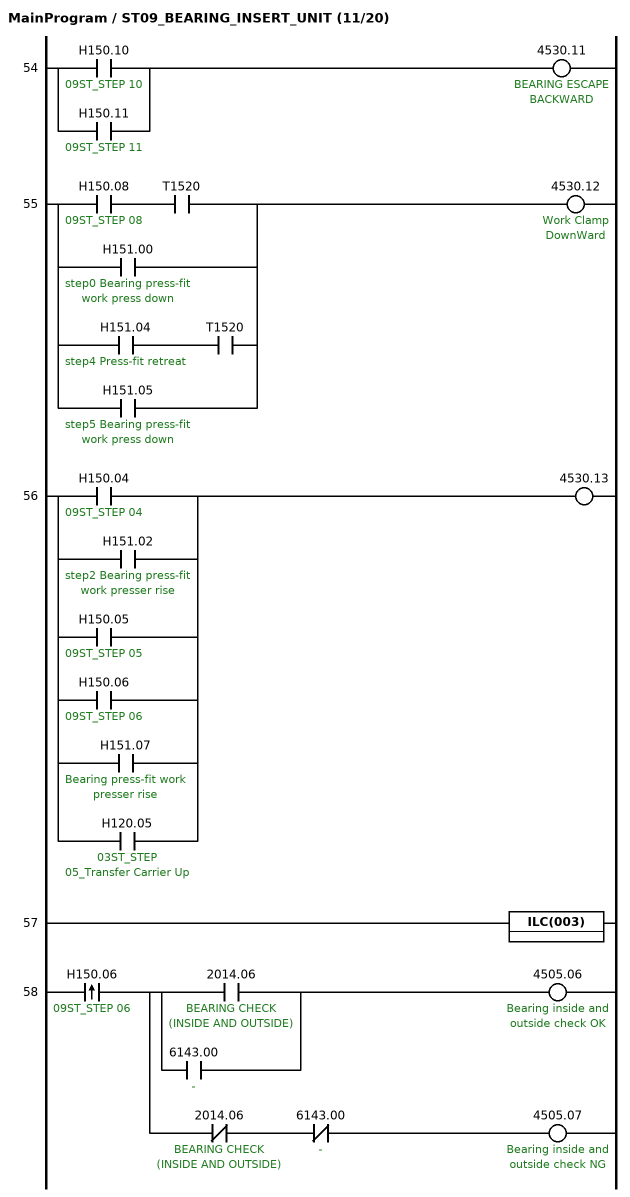
; rung 54
LD H150.10  ; 09ST_STEP 10
OR H150.11  ; 09ST_STEP 11
OUT 4530.11  ; BEARING ESCAPE BACKWARD
; rung 55
LD H150.08  ; 09ST_STEP 08
AND T1520
OR H151.00  ; step0 Bearing press-fit work press down
LD H151.04  ; step4 Press-fit retreat
AND T1520
ORLD
OR H151.05  ; step5 Bearing press-fit work press down
OUT 4530.12  ; Work Clamp DownWard
; rung 56
LD H150.04  ; 09ST_STEP 04
OR H151.02  ; step2 Bearing press-fit work presser rise
OR H150.05  ; 09ST_STEP 05
OR H150.06  ; 09ST_STEP 06
OR H151.07  ; Bearing press-fit work presser rise
OR H120.05  ; 03ST_STEP 05_Transfer Carrier Up
OUT 4530.13
; rung 57
ILC(003)
; rung 58
@LD H150.06  ; 09ST_STEP 06
OUT TR0
LD 2014.06  ; BEARING CHECK (INSIDE AND OUTSIDE)
OR 6143.00  ; -
ANDLD
OUT 4505.06  ; Bearing inside and outside check OK
LD TR0
ANDNOT 2014.06  ; BEARING CHECK (INSIDE AND OUTSIDE)
ANDNOT 6143.00  ; -
OUT 4505.07  ; Bearing inside and outside check NG

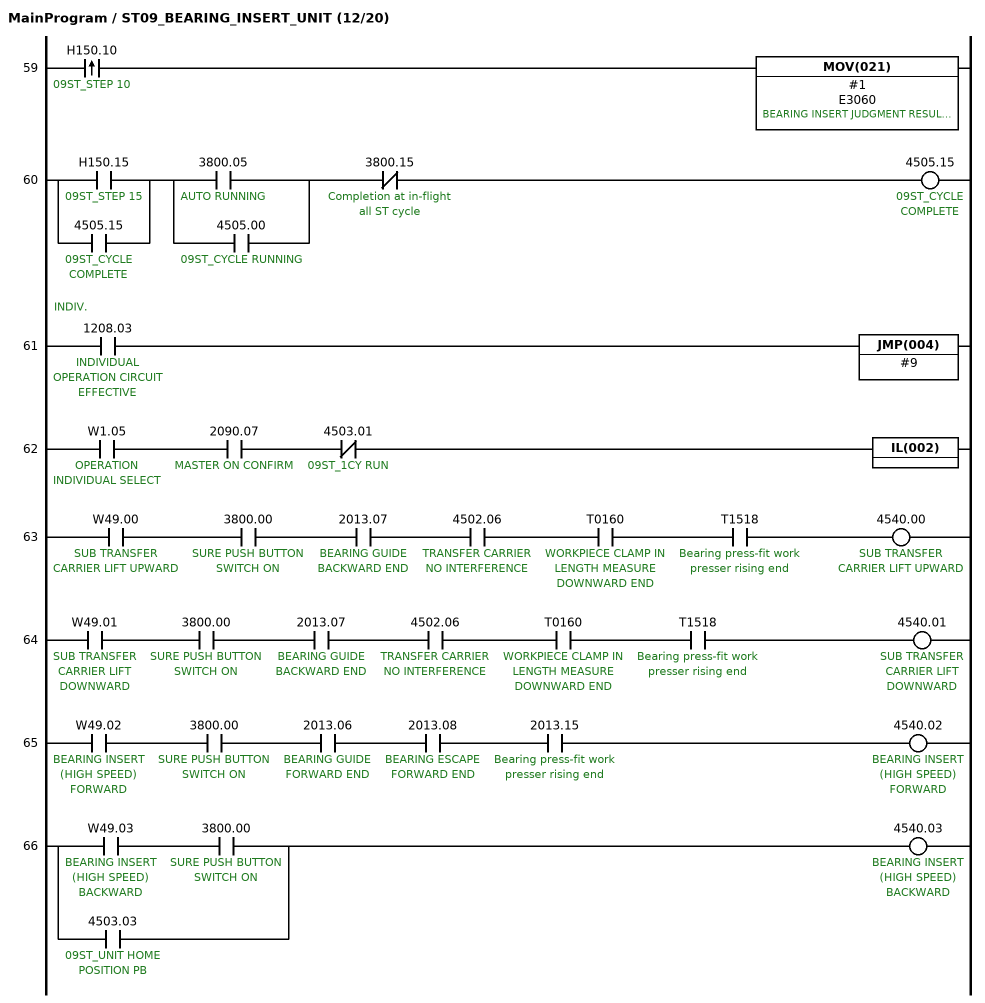
; rung 59
@LD H150.10  ; 09ST_STEP 10
MOV(021) #1 E3060  ; BEARING INSERT JUDGMENT RESULT (1:OK,2:NG)
; rung 60
LD H150.15  ; 09ST_STEP 15
OR 4505.15  ; 09ST_CYCLE COMPLETE
LD 3800.05  ; AUTO RUNNING
OR 4505.00  ; 09ST_CYCLE RUNNING
ANDLD
ANDNOT 3800.15  ; Completion at in-flight all ST cycle
OUT 4505.15  ; 09ST_CYCLE COMPLETE
; rung 61: INDIV.
LD 1208.03  ; INDIVIDUAL OPERATION CIRCUIT EFFECTIVE
JMP(004) #9
; rung 62
LD W1.05  ; OPERATION INDIVIDUAL SELECT
AND 2090.07  ; MASTER ON CONFIRM
ANDNOT 4503.01  ; 09ST_1CY RUN
IL(002)
; rung 63
LD W49.00  ; SUB TRANSFER CARRIER LIFT UPWARD
AND 3800.00  ; SURE PUSH BUTTON SWITCH ON
AND 2013.07  ; BEARING GUIDE BACKWARD END
AND 4502.06  ; TRANSFER CARRIER NO INTERFERENCE
AND T0160  ; WORKPIECE CLAMP IN LENGTH MEASURE DOWNWARD END
AND T1518  ; Bearing press-fit work presser rising end
OUT 4540.00  ; SUB TRANSFER CARRIER LIFT UPWARD
; rung 64
LD W49.01  ; SUB TRANSFER CARRIER LIFT DOWNWARD
AND 3800.00  ; SURE PUSH BUTTON SWITCH ON
AND 2013.07  ; BEARING GUIDE BACKWARD END
AND 4502.06  ; TRANSFER CARRIER NO INTERFERENCE
AND T0160  ; WORKPIECE CLAMP IN LENGTH MEASURE DOWNWARD END
AND T1518  ; Bearing press-fit work presser rising end
OUT 4540.01  ; SUB TRANSFER CARRIER LIFT DOWNWARD
; rung 65
LD W49.02  ; BEARING INSERT (HIGH SPEED) FORWARD
AND 3800.00  ; SURE PUSH BUTTON SWITCH ON
AND 2013.06  ; BEARING GUIDE FORWARD END
AND 2013.08  ; BEARING ESCAPE FORWARD END
AND 2013.15  ; Bearing press-fit work presser rising end
OUT 4540.02  ; BEARING INSERT (HIGH SPEED) FORWARD
; rung 66
LD W49.03  ; BEARING INSERT (HIGH SPEED) BACKWARD
AND 3800.00  ; SURE PUSH BUTTON SWITCH ON
OR 4503.03  ; 09ST_UNIT HOME POSITION PB
OUT 4540.03  ; BEARING INSERT (HIGH SPEED) BACKWARD

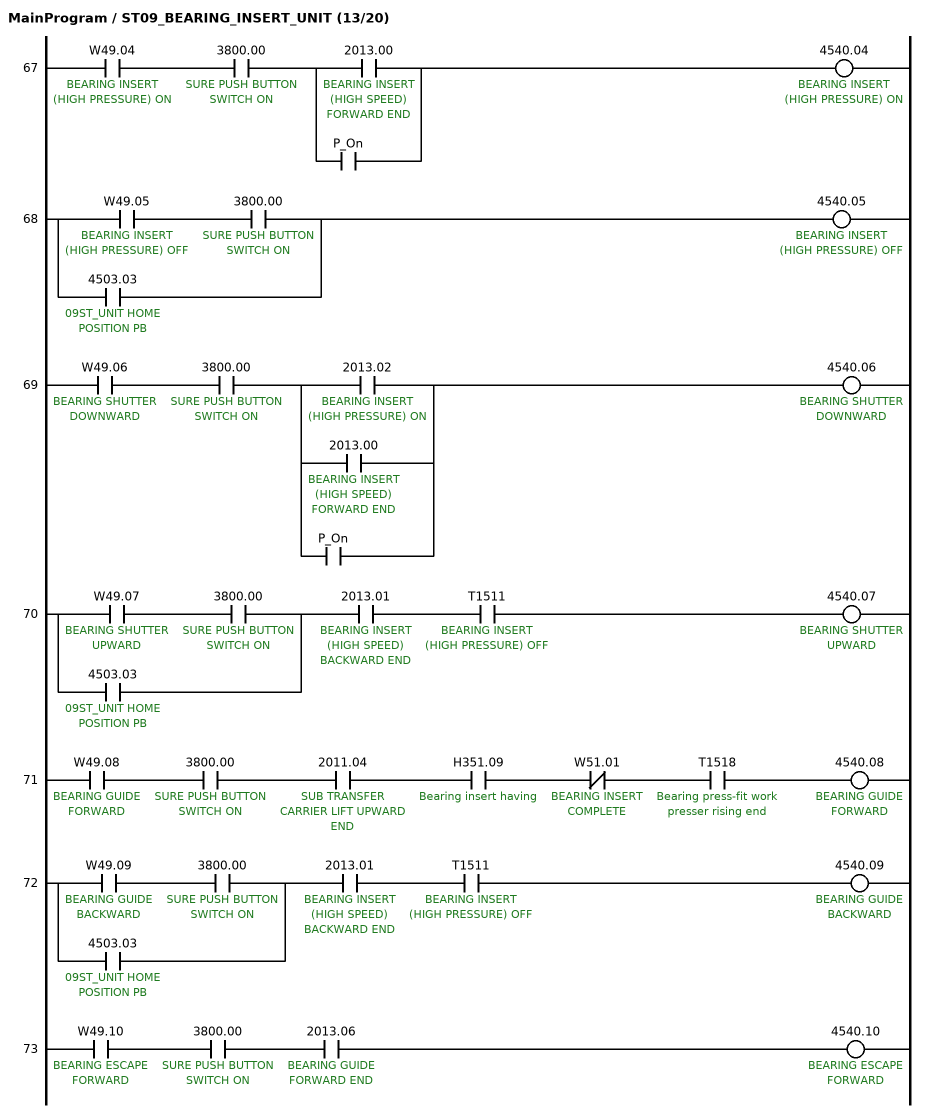
; rung 67
LD W49.04  ; BEARING INSERT (HIGH PRESSURE) ON
AND 3800.00  ; SURE PUSH BUTTON SWITCH ON
LD 2013.00  ; BEARING INSERT (HIGH SPEED) FORWARD END
OR P_On
ANDLD
OUT 4540.04  ; BEARING INSERT (HIGH PRESSURE) ON
; rung 68
LD W49.05  ; BEARING INSERT (HIGH PRESSURE) OFF
AND 3800.00  ; SURE PUSH BUTTON SWITCH ON
OR 4503.03  ; 09ST_UNIT HOME POSITION PB
OUT 4540.05  ; BEARING INSERT (HIGH PRESSURE) OFF
; rung 69
LD W49.06  ; BEARING SHUTTER DOWNWARD
AND 3800.00  ; SURE PUSH BUTTON SWITCH ON
LD 2013.02  ; BEARING INSERT (HIGH PRESSURE) ON
OR 2013.00  ; BEARING INSERT (HIGH SPEED) FORWARD END
OR P_On
ANDLD
OUT 4540.06  ; BEARING SHUTTER DOWNWARD
; rung 70
LD W49.07  ; BEARING SHUTTER UPWARD
AND 3800.00  ; SURE PUSH BUTTON SWITCH ON
OR 4503.03  ; 09ST_UNIT HOME POSITION PB
AND 2013.01  ; BEARING INSERT (HIGH SPEED) BACKWARD END
AND T1511  ; BEARING INSERT (HIGH PRESSURE) OFF
OUT 4540.07  ; BEARING SHUTTER UPWARD
; rung 71
LD W49.08  ; BEARING GUIDE FORWARD
AND 3800.00  ; SURE PUSH BUTTON SWITCH ON
AND 2011.04  ; SUB TRANSFER CARRIER LIFT UPWARD END
AND H351.09  ; Bearing insert having
ANDNOT W51.01  ; BEARING INSERT COMPLETE
AND T1518  ; Bearing press-fit work presser rising end
OUT 4540.08  ; BEARING GUIDE FORWARD
; rung 72
LD W49.09  ; BEARING GUIDE BACKWARD
AND 3800.00  ; SURE PUSH BUTTON SWITCH ON
OR 4503.03  ; 09ST_UNIT HOME POSITION PB
AND 2013.01  ; BEARING INSERT (HIGH SPEED) BACKWARD END
AND T1511  ; BEARING INSERT (HIGH PRESSURE) OFF
OUT 4540.09  ; BEARING GUIDE BACKWARD
; rung 73
LD W49.10  ; BEARING ESCAPE FORWARD
AND 3800.00  ; SURE PUSH BUTTON SWITCH ON
AND 2013.06  ; BEARING GUIDE FORWARD END
OUT 4540.10  ; BEARING ESCAPE FORWARD

